FUNCTION_BLOCK FB_CoE_BYTE EXTENDS FB_CoE_Base
(* 
   FB_init:
	(	ipCoeConnection := fbCoeConnection, (*each EC-Slave needs one FB_CoE_Connection*)
		nIndex     		:= 16#8010, (* CoE Object Index *)
		nSubIndex  		:= 16#11 (* Subindex of CoE Object *));
 *)
VAR
	{attribute 'hide'}
	nValue : BYTE;
END_VAR

PROPERTY PROTECTED cbBufLen : UDINT
GET
cbBufLen := SIZEOF(nValue);
END_GET
END_PROPERTY

PROPERTY PROTECTED pSrcBuf : PVOID
GET
pSrcBuf := ADR(nValue);
END_GET
END_PROPERTY

{attribute 'monitoring':='call'}
PROPERTY Value : BYTE
GET
Value := nValue;
END_GET
SET
nValue := Value;

//Trigger a new write cycle
THIS^.bWriteDone 	:= FALSE;
END_SET
END_PROPERTY

END_FUNCTION_BLOCK

(* stored: Version 1.1.0.1, ProductVersion 3.1.4024.12
   POU FB_CoE_BYTE: Id {13617f42-f0fc-4b81-ae0a-db569bfca0cf}, SpecialFunc None
   Property cbBufLen: Id {bb987054-92e8-4fd2-a1ee-725bd2adcf78}
   Get Get: Id {ffb6eb91-ed8f-4925-ad4c-52b4b217ae0b}
   Property pSrcBuf: Id {2624f113-aa55-43f2-acac-73bc58fc817f}
   Get Get: Id {bca286ec-768b-463a-bbeb-478804d46602}
   Property Value: Id {6b423d12-a074-47ca-be33-f5ead9938711}
   Get Get: Id {48bfc861-d82e-414e-85ed-6a125bb84d3b}
   Set Set: Id {bd5a8ef5-5b5d-4596-9d6e-be125b9ec5a4} *)
